PROGRAM MAIN
VAR
	// trigger command execution for Telegram samples
	bGetTelegram					: BOOL;

	fbHttpClientTelegram			: FB_IotHttpClient :=(sHostName := 'api.telegram.org',
									bKeepAlive := FALSE, tConnectionTimeout := T#10S);

	fbHttpGetTelegram				: FB_TestHTTP_Get_Telegram;
	sMessage						: STRING(500) := 'Hello from TwinCAT';
END_VAR

// init client parameters at startup
IF NOT fbHttpClientTelegram.bConfigured THEN
	fbHttpClientTelegram.nHostPort := 443;
	fbHttpClientTelegram.stTLS.bNoServerCertCheck := TRUE;
END_IF

IF fbHttpClientTelegram.bConfigured THEN
	fbHttpGetTelegram(bSend := bGetTelegram, fbClient := fbHttpClientTelegram, sMessage := sMessage);
END_IF

fbHttpClientTelegram.Execute();

END_PROGRAM

(* stored: Version 1.1.0.1, ProductVersion 3.1.4024.6
   POU MAIN: Id {6d4237ee-1c29-4d23-9e91-4101e71768e5}, SpecialFunc None *)
